TYPE ST_CasePackerInfo :	(* 8 bytes *)
STRUCT
	ProductionSite 	: STRING(4);
	ProductionLine 	: STRING(4);
END_STRUCT
END_TYPE

(* stored: Version 1.1.0.1, ProductVersion 3.1.4024.15
   DUT ST_CasePackerInfo: Id {8d236e61-07ba-4fcb-ac04-03c5560ea14e} *)
